{attribute 'linkalways'} 
{attribute 'no_explicit_call' := 'This FB is a CLASS and must be accessed using methods or properties'}
{attribute 'enable_dynamic_creation'}
FUNCTION_BLOCK _ETcVnContoursMatchComparisonMethod EXTENDS EnumDatatypeBase
VAR
	localData : ETcVnContoursMatchComparisonMethod;
	activeData : REFERENCE TO ETcVnContoursMatchComparisonMethod;
	enumBaseDatatype : _DINT(localData);
END_VAR

METHOD PRIVATE AddLocalEnumeration
VAR_INPUT
	Enumeration : T_MAXSTRING;
	Value : ETcVnContoursMatchComparisonMethod;
END_VAR
AddEnumeration(Enumeration, Value);
END_METHOD

PROPERTY PUBLIC Address : PVOID
GET
Address := ADR(activeData);
END_GET
END_PROPERTY

METHOD PUBLIC ClearReference
VAR_INPUT
END_VAR
activeData REF= localData;
SetBaseDatatypeReference();
END_METHOD

METHOD PUBLIC Clone : I_Datatype
VAR
    pClone : POINTER TO _ETcVnContoursMatchComparisonMethod;
END_VAR
pClone := __NEW(_ETcVnContoursMatchComparisonMethod(InitialValue := Value));
Clone := pClone^;
END_METHOD

METHOD FB_init : BOOL
VAR_INPUT
	bInitRetains : BOOL; // if TRUE, the retain variables are initialized (warm start / cold start)
	bInCopyCode : BOOL;  // if TRUE, the instance afterwards gets moved into the copy code (online change)
	InitialValue : ETcVnContoursMatchComparisonMethod;
END_VAR
localData := InitialValue;
AddBaseDatatype(enumBaseDatatype);
ClearReference();

AddLocalEnumeration('TCVN_CMCM_CONTOURS_MATCH_I1', ETcVnContoursMatchComparisonMethod.TCVN_CMCM_CONTOURS_MATCH_I1);
AddLocalEnumeration('TCVN_CMCM_CONTOURS_MATCH_I2', ETcVnContoursMatchComparisonMethod.TCVN_CMCM_CONTOURS_MATCH_I2);
AddLocalEnumeration('TCVN_CMCM_CONTOURS_MATCH_I3', ETcVnContoursMatchComparisonMethod.TCVN_CMCM_CONTOURS_MATCH_I3);
END_METHOD

PROPERTY PUBLIC Identifier : T_MAXSTRING
GET
Identifier := 'ETcVnContoursMatchComparisonMethod';
END_GET
END_PROPERTY

METHOD IsEnumeratorValueEqual : BOOL
VAR_INPUT
	Enumerator : I_KeyValueForwardEnumerator;
END_VAR
VAR
	storedValue : ETcVnContoursMatchComparisonMethod;
END_VAR
IF NOT Enumerator.TryGet(storedValue) THEN
	RETURN;
END_IF

IsEnumeratorValueEqual := storedValue = activeData;
END_METHOD

METHOD PUBLIC MakeReferenceTo
VAR_INPUT
	ReferenceTarget : REFERENCE TO ETcVnContoursMatchComparisonMethod;
END_VAR
activeData REF= ReferenceTarget;
SetBaseDatatypeReference();
END_METHOD

METHOD PROTECTED SetBaseDatatypeReference
VAR_INPUT
END_VAR
enumBaseDatatype.MakeReferenceTo(activeData);
END_METHOD

PROPERTY PUBLIC Size : UDINT
GET
Size := SIZEOF(activeData);
END_GET
END_PROPERTY

METHOD TryMakeReferenceTo : BOOL
VAR_INPUT
	Target : I_Datatype;
END_VAR
VAR
	targetAsEnum : I_EnumDatatype;
	pTargetData : POINTER TO ETcVnContoursMatchComparisonMethod;
END_VAR
IF NOT Target.TryResolveAsEnumDatatype(targetAsEnum) THEN
	RETURN;
END_IF

IF targetAsEnum.Identifier <> Identifier THEN
	RETURN;
END_IF

pTargetData := Target.Address;
activeData REF= pTargetData^;
SetBaseDatatypeReference();
TryMakeReferenceTo := TRUE;
END_METHOD

PROPERTY PUBLIC Value : ETcVnContoursMatchComparisonMethod
GET
Value := activeData;
END_GET
SET
activeData := Value;
END_SET
END_PROPERTY

END_FUNCTION_BLOCK

(* stored: Version 1.1.0.1, ProductVersion 3.1.4024.12
   POU _ETcVnContoursMatchComparisonMethod: Id {f92bf982-4b2f-064d-27bb-a035a08125e4}, SpecialFunc None
   Folder Constructor: Id {d97a65b0-1915-0b68-28d6-bc38c6451ad9}
   Folder Private: Id {bebc5086-3c88-00bf-0ff1-ed32781a934b}
   Folder Protected: Id {17a66745-395d-08c8-2aad-c76fd1f5c654}
   Method AddLocalEnumeration: Id {30c0f396-4070-0b00-3193-62391a60a069}
   Property Address: Id {dbedb1d2-2bc9-0528-361d-439d3a5ffee4}
   Get Get: Id {f820c8ee-7363-0447-0ee6-85dce0a0b2f3}
   Method ClearReference: Id {f929c31c-6eea-0d84-1f30-578969b6c05b}
   Method Clone: Id {d401cee9-83d2-09c1-36d0-00f524c3e2d5}
   Method FB_init: Id {fa605eeb-c1a5-0357-0761-e76787a19270}
   Property Identifier: Id {59782c08-feff-08ea-213d-66dcc7c14d36}
   Get Get: Id {9ffc41e0-4470-07b7-3e92-3b962610aa23}
   Method IsEnumeratorValueEqual: Id {7618762a-446f-087e-25ce-ffaf5fb5d5e3}
   Method MakeReferenceTo: Id {a6fcea3d-74c9-0f71-0341-03b77ae5ed11}
   Method SetBaseDatatypeReference: Id {d24ab8c4-a2c0-034d-311d-caa5d682a0e9}
   Property Size: Id {089ed319-4d17-0b8c-332d-453d231a75b7}
   Get Get: Id {9359e1bb-4a1b-0edc-0ba5-80c5699a70d0}
   Method TryMakeReferenceTo: Id {ee7f5c35-fd4a-09fa-217b-b7f5baf7f6b3}
   Property Value: Id {6c6649e6-8347-0575-08e8-b07f60088e8b}
   Get Get: Id {2da7d5d7-e154-0bf9-2f66-25919bccd469}
   Set Set: Id {ba9c4b2d-ab1f-0b49-3ebf-076a17215e8e} *)
